Universal Robots PolyScope program: washer_release.urp

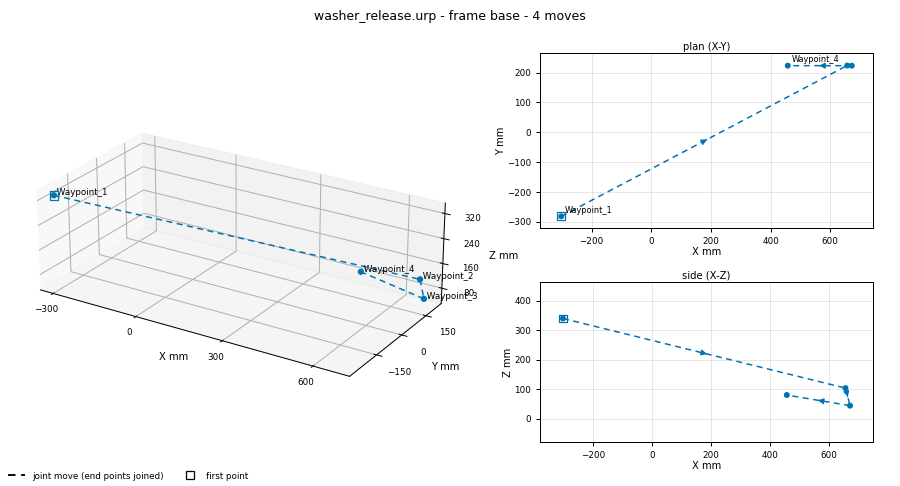
[picture p0: tool path of washer_release.urp in frame base, 4 of 4 moves have a stored position in this frame; points joined in program order, loops and branches not executed]
Program washer_release (installation=default directory=/programs createdIn=5.9.5.1031259 lastSavedIn=5.9.5.1031259 robotSerialNumber=20215500597)
Calibrated DH parameters: a=[0.000193, -0.066673, -0.391568, -0.000012, 0.00005, 0]; d=[0.162643, -472.05677, 465.132521, 7.058239, 0.099746, 0.099582]; alpha=[1.571116, 0.00089, 0.003862, 1.569269, -1.569248, 0]; deltaTheta=[0, -1.413394, 7.628392, 0.068187, 0, -0.000001]
Robot Program (runOnlyOnce=false)
  MoveJ speed 60 deg/s, acceleration 80 deg/s^2 (useActiveTCP=true) feature=Base
    Waypoint Waypoint_1: TCP in base x=-301.653 y=-281.559 z=339.218 mm, rx=1.1718 ry=-1.2853 rz=1.2611 rad; joints [331.698, -104.001, 123.671, 339.069, -27.886, -263.998] deg; TCP offset x=0 y=0 z=191.5 mm, rx=0 ry=0 rz=0 rad
    Waypoint Waypoint_2: TCP in base x=656.517 y=223.841 z=103.164 mm, rx=-0.0395 ry=1.5513 rz=-0.0092 rad; joints [192.488, -61.382, 120.953, 299.229, 101.514, -92.016] deg
    Waypoint Waypoint_3: TCP in base x=671.899 y=223.323 z=43.584 mm, rx=-0.0517 ry=1.642 rz=-0.0273 rad; joints [192.188, -55.049, 117.199, 301.971, 101.525, -91.992] deg
    URCap Gripper (Robotiq_Grippers, Robotiq Inc.) dataModel(position=0.0, force=40.0, speed=49.80392156862745, positionInDouble=0.0, forceInDouble=40.0, speedInDouble=49.80392156862745, slaveIds=[9], blocking=true)
    Waypoint Waypoint_4: TCP in base x=457.414 y=223.392 z=79.648 mm, rx=-0.0044 ry=1.6521 rz=-0.0401 rad; joints [205.889, -73.3, 142.656, 295.77, 117.318, -89.324] deg
    Halt
